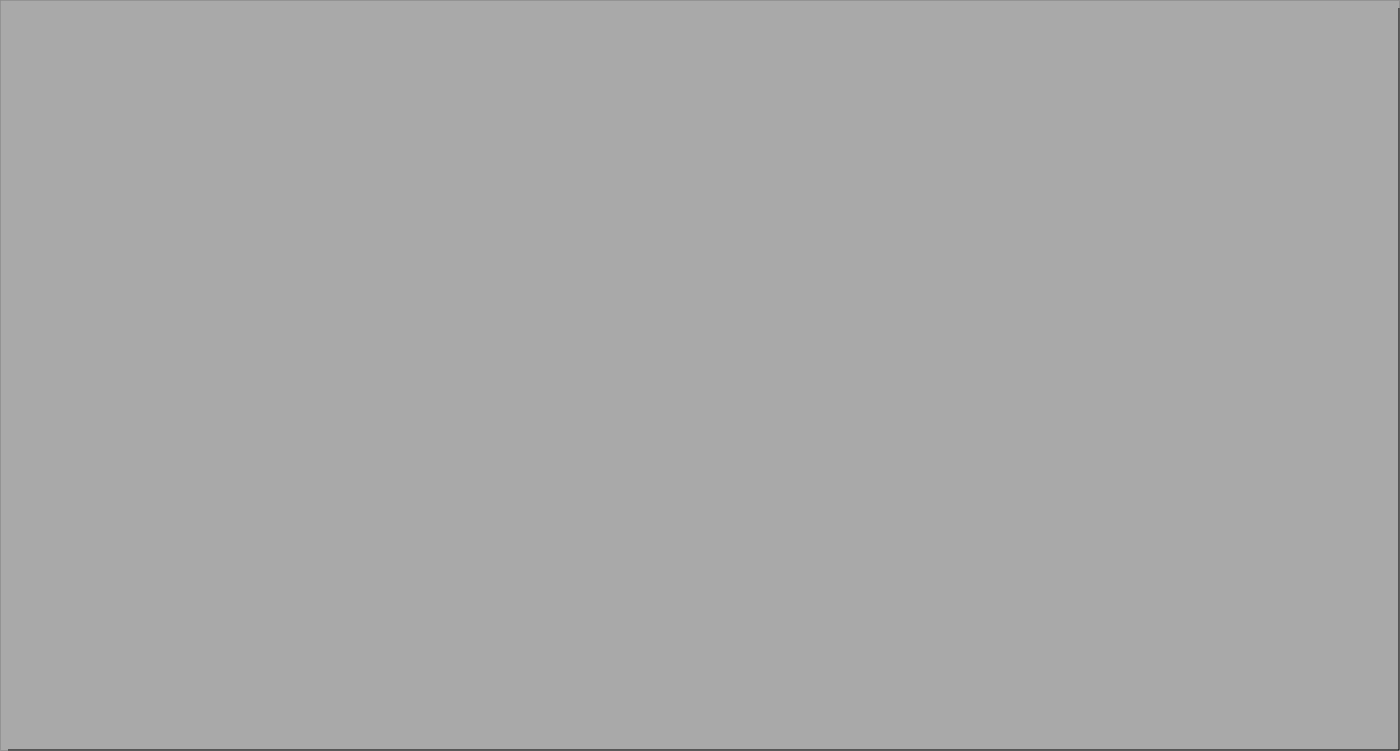
VISUALIZATION PID_alt  // 1792x962, background image 
    Rectangle (10,960 1780x2)
    Rectangle (1790,10 2x950)
END_VISUALIZATION

(* stored: Version 1.1.0.1, ProductVersion 3.1.4024.3
   Visu PID_alt: Id {a5002a3b-dba4-4ba7-bba7-5b0179552df0} *)
